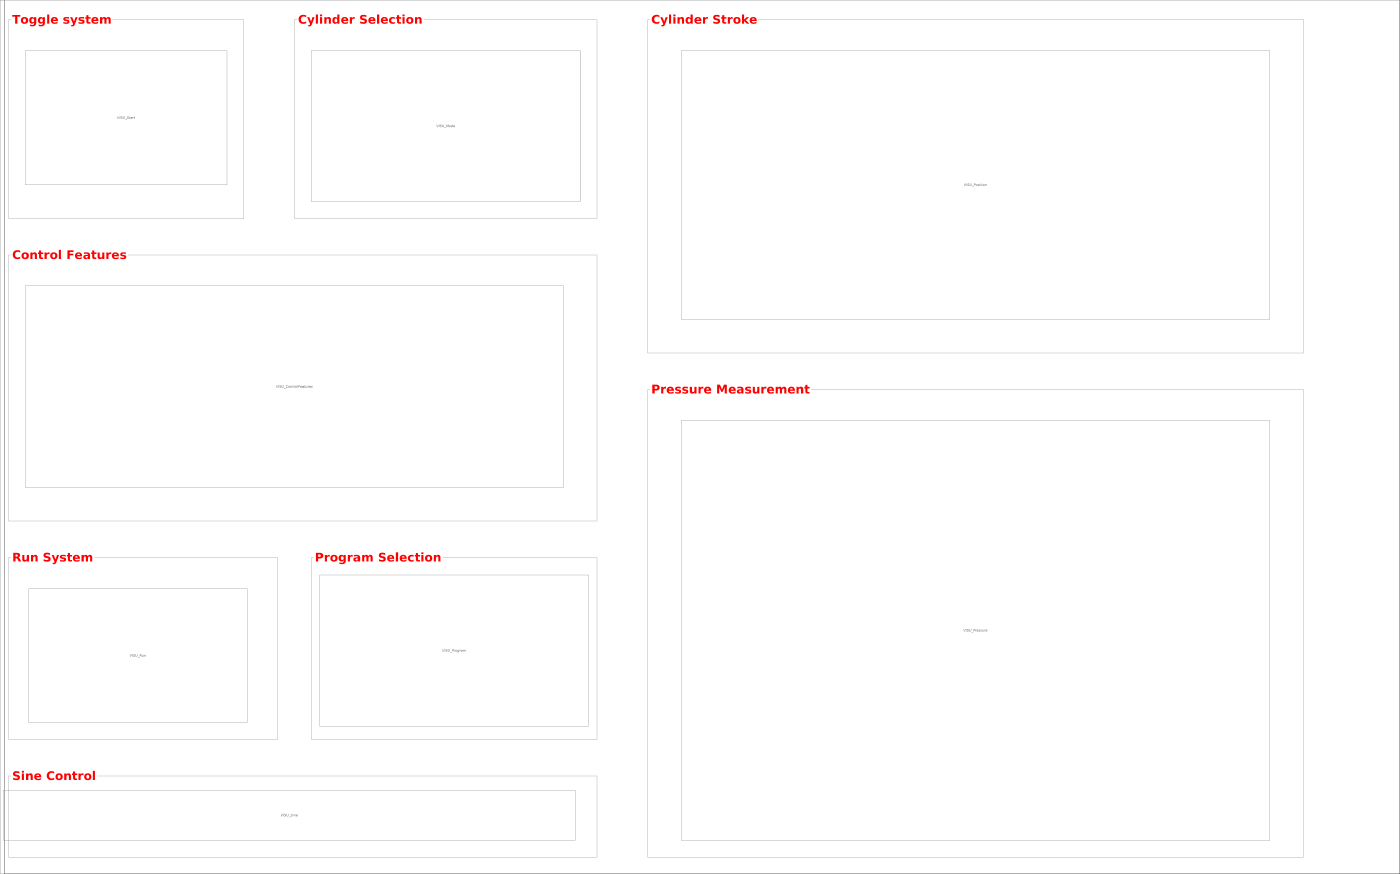
VISUALIZATION Visualization  // 4162x2600
    Rectangle (12,0 4150x2600)
    GroupBox (25,750 1750x800), "Control Features"
    GroupBox (25,50 700x600), "Toggle system"
    GroupBox (925,1650 850x550), "Program Selection"
    GroupBox (1925,1150 1950x1400), "Pressure Measurement"
    GroupBox (25,1650 800x550), "Run System"
        Frame (925,60 800x450)
            shows VISU_Program()
        Frame (60,100 650x400)
            shows VISU_Run()
    GroupBox (875,50 900x600), "Cylinder Selection"
    GroupBox (1925,50 1950x1000), "Cylinder Stroke"
    Frame (75,150 600x400)
        shows VISU_Start()
    Frame (2025,150 1750x800)
        shows VISU_Position()
    Frame (2025,1250 1750x1250)
        shows VISU_Pressure()
    Frame (75,850 1600x600)
        shows VISU_ControlFeatures()
    Frame (925,150 800x450)
        shows VISU_Mode()
    GroupBox (25,2300 1750x250), "Sine Control"
    Frame (10,2350 1700x150)
        shows VISU_Sine()
END_VISUALIZATION

(* stored: Version 1.1.0.1
   Visu Visualization: Id {d7aa0e2f-c517-48a7-8af6-49fcb84800c2} *)
